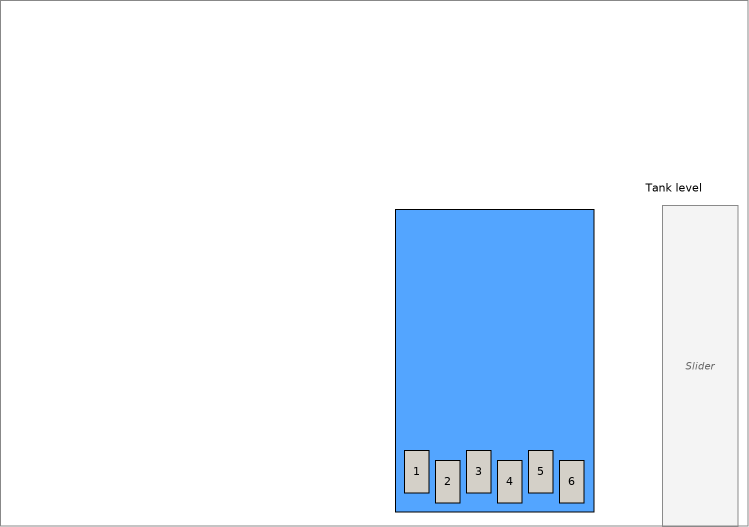
VISUALIZATION Visualization  // 749x527
    Rectangle (395,209 199x303)
    RoundedRectangle (404,450 25x43), "1", colour toggle: MAIN.PumpTank.PumpsArray[1].RunState=PumpState.RUN
    RoundedRectangle (435,460 25x43), "2", colour toggle: MAIN.PumpTank.PumpsArray[2].RunState=PumpState.RUN
    RoundedRectangle (466,450 25x43), "3", colour toggle: MAIN.PumpTank.PumpsArray[3].RunState=PumpState.RUN
    RoundedRectangle (497,460 25x43), "4", colour toggle: MAIN.PumpTank.PumpsArray[4].RunState=PumpState.RUN
    RoundedRectangle (559,460 25x43), "6", colour toggle: MAIN.PumpTank.PumpsArray[6].RunState=PumpState.RUN
    RoundedRectangle (528,450 25x43), "5", colour toggle: MAIN.PumpTank.PumpsArray[5].RunState=PumpState.RUN
    Slider (662,205 76x322), variable: MAIN.PumpTank.Level, scale 0..1000
    Label (599,173 150x30), "Tank level"
END_VISUALIZATION

(* stored: Version 1.1.0.1, ProductVersion 3.1.4024.15
   Visu Visualization: Id {0647d19e-d6e0-46f8-9f57-c867682fef48} *)
